TYPE U_Data :
UNION
	
	rxtxBuffer       : ARRAY[0..255] OF BYTE;
	sText : STRING;
	
END_UNION
END_TYPE

(* stored: Version 1.1.0.1
   DUT U_Data: Id {ec03eef9-722c-401d-9919-04e50c633c84} *)
